{attribute 'qualified_only'}
VAR_GLOBAL
	amsNetId : T_AmsNetId  := '';
END_VAR

(* stored: Version 1.1.0.1, ProductVersion 3.1.4024.11
   GVL GVL: Id {010dfc94-3f13-4598-ad85-5aa8eec9bf3c} *)
